FUNCTION F_SINT_RTN : SINT
VAR_INPUT
	stArg : ST_Arg;
END_VAR
VAR
	sysVar_Info : __SYSTEM.VAR_INFO;
END_VAR

sysVar_Info := __VARINFO(F_SINT_RTN);
IF stArg.TypeClass = sysVar_Info.TypeClass THEN 
	F_SINT_RTN := TO_SINT(stArg.sValue);
	END_IF

END_FUNCTION

(* stored: Version 1.1.0.1, ProductVersion 3.1.4024.4
   POU F_SINT_RTN: Id {94ae68cf-d1fa-4a20-8204-2d92578bf740}, SpecialFunc None *)
